TYPE E_2OO3_MODE :
(
	MODE_2OO3 := 0,
	IG_CH1 := 1,
	IG_CH2 := 2,
	IG_CH3 := 3
);
END_TYPE

(* stored: Version 1.1.0.1, ProductVersion 3.1.4022.18
   DUT E_2OO3_MODE: Id {7da80cf0-4fde-4ce3-82c4-7c1c74badc27} *)
